TYPE DUT_AxisStatus_v0_01:
STRUCT
    bEnable: BOOL;
    bReset: BOOL;
    bExecute: BOOL;
    nCommand: UINT;
    nCmdData: UINT;
    fVelocity: LREAL;
    fPosition: LREAL;
    fAcceleration: LREAL;
    fDeceleration: LREAL;
    bJogFwd: BOOL;
    bJogBwd: BOOL;
    bLimitFwd: BOOL;
    bLimitBwd: BOOL;
    fOverride: LREAL:=100;
    bHomeSensor: BOOL;
    bEnabled: BOOL;
    bError: BOOL;
    nErrorId: UDINT;
    fActVelocity: LREAL;
    fActPosition: LREAL;
    fActDiff: LREAL;
    bHomed:BOOL;
    bBusy:BOOL;
END_STRUCT
END_TYPE

(* stored: Version 1.1.0.1, ProductVersion 3.1.4024.0
   DUT DUT_AxisStatus_v0_01: Id {c6013052-aa22-40c3-8a00-8a16922e6eac} *)
